PROGRAM RemovalProgram
VAR
END_VAR

// Written 25.8.2023 by Daniel Kelly

// The purpose of this POU is to automate the emptying of the system
//OpenValves will open both top and bottom valves
//RemovalMotorON will turn on the removal motor
//FM1_ON turns on the grey feeding motor M1
// The steps OFF1, OFF2 etc. turns of the removal motor and both top and bottom valves

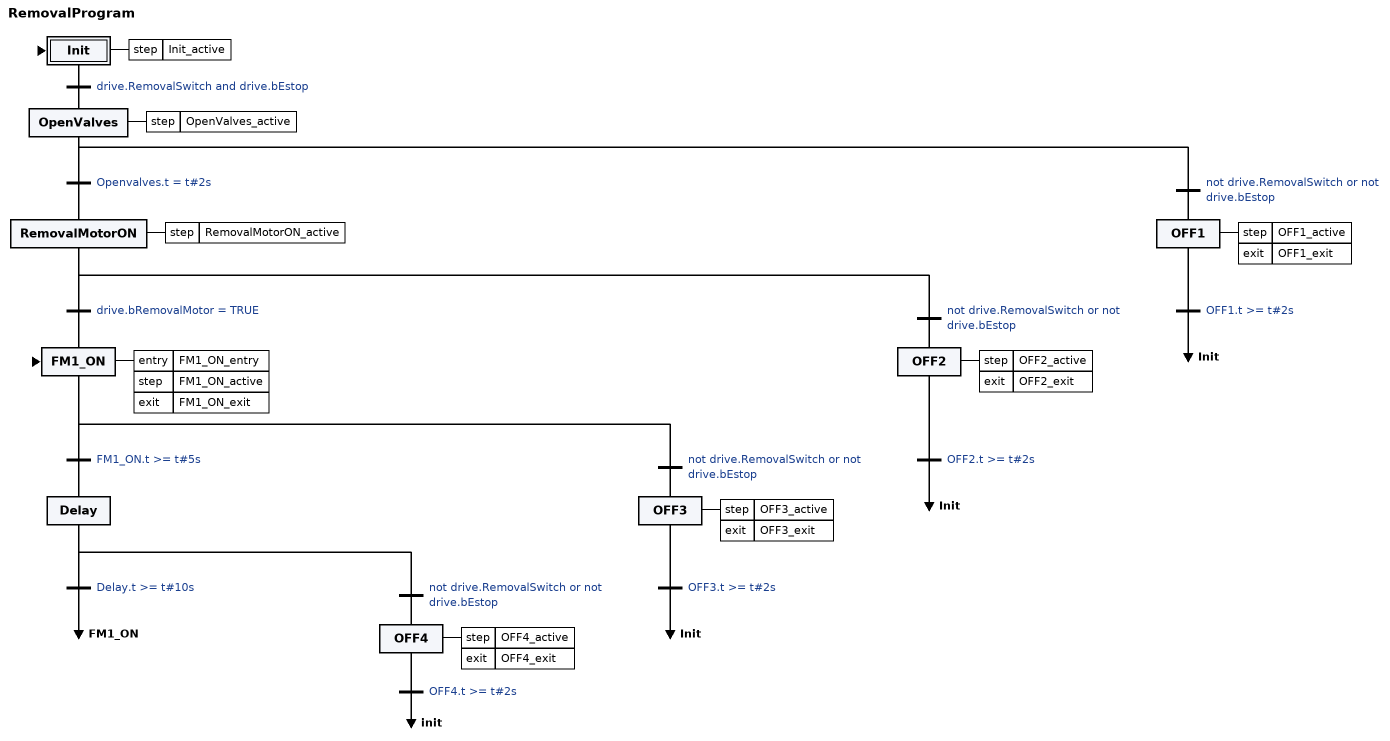
INITIAL_STEP Init:
    Init_active(N);  // step action
END_STEP
TRANSITION FROM Init TO OpenValves
    := drive.RemovalSwitch and drive.bEstop;
END_TRANSITION
STEP OpenValves:
    OpenValves_active(N);  // step action
END_STEP
TRANSITION FROM OpenValves TO RemovalMotorON
    := Openvalves.t = t#2s;
END_TRANSITION
TRANSITION FROM OpenValves TO OFF1
    := not drive.RemovalSwitch or not drive.bEstop;
END_TRANSITION
STEP OFF1:
    OFF1_active(N);  // step action
    OFF1_exit(P0);  // exit action
END_STEP
TRANSITION FROM OFF1 TO Init
    := OFF1.t >= t#2s;
END_TRANSITION
STEP RemovalMotorON:
    RemovalMotorON_active(N);  // step action
END_STEP
TRANSITION FROM RemovalMotorON TO FM1_ON
    := drive.bRemovalMotor = TRUE;
END_TRANSITION
TRANSITION FROM RemovalMotorON TO OFF2
    := not drive.RemovalSwitch or not drive.bEstop;
END_TRANSITION
STEP OFF2:
    OFF2_active(N);  // step action
    OFF2_exit(P0);  // exit action
END_STEP
TRANSITION FROM OFF2 TO Init
    := OFF2.t >= t#2s;
END_TRANSITION
STEP FM1_ON:
    FM1_ON_entry(P1);  // entry action
    FM1_ON_active(N);  // step action
    FM1_ON_exit(P0);  // exit action
END_STEP
TRANSITION FROM FM1_ON TO Delay
    := FM1_ON.t >= t#5s;
END_TRANSITION
TRANSITION FROM FM1_ON TO OFF3
    := not drive.RemovalSwitch or not drive.bEstop;
END_TRANSITION
STEP OFF3:
    OFF3_active(N);  // step action
    OFF3_exit(P0);  // exit action
END_STEP
TRANSITION FROM OFF3 TO Init
    := OFF3.t >= t#2s;
END_TRANSITION
STEP Delay:
END_STEP
TRANSITION FROM Delay TO FM1_ON
    := Delay.t >= t#10s;
END_TRANSITION
TRANSITION FROM Delay TO OFF4
    := not drive.RemovalSwitch or not drive.bEstop;
END_TRANSITION
STEP OFF4:
    OFF4_active(N);  // step action
    OFF4_exit(P0);  // exit action
END_STEP
TRANSITION FROM OFF4 TO init
    := OFF4.t >= t#2s;
END_TRANSITION

ACTION FM1_ON_active:
IF drive.ATV_TPDO_Input1_Status_Word = atv_status.rdy2SwitchON THEN 
	drive.ATV_RPDO_Output1_Control_Word := 7;
END_IF

IF drive.ATV_TPDO_Input1_Status_Word = atv_status.SwitchedON THEN 
	drive.ATV_RPDO_Output1_Control_Word := 15;
	
END_IF

drive.bM1active := TRUE;
END_ACTION

ACTION FM1_ON_entry:
drive.ATV_RPDO_Output2_Target_Velocity := 1000;
drive.ATV_RPDO_Output1_Control_Word := 6;
END_ACTION

ACTION FM1_ON_exit:
drive.ATV_RPDO_Output1_Control_Word := 7; 
drive.bM1active := FALSE;
END_ACTION

ACTION Init_active:

END_ACTION

ACTION OFF1_active:
drive.bRemovalMotor := FALSE;
drive.CloseTopValve := TRUE;
drive.CloseBottomValve := TRUE;

drive.OpenTopValve := FALSE;
drive.OpenBottomValve := FALSE;

drive.bValveLamp := FALSE;
END_ACTION

ACTION OFF1_exit:
drive.CloseBottomValve := FALSE;
drive.CloseTopValve := FALSE;
END_ACTION

ACTION OFF2_active:
drive.bRemovalMotor := FALSE;
drive.CloseTopValve := TRUE;
drive.CloseBottomValve := TRUE;

drive.OpenTopValve := FALSE;
drive.OpenBottomValve := FALSE;

drive.bValveLamp := FALSE;
END_ACTION

ACTION OFF2_exit:
drive.CloseBottomValve := FALSE;
drive.CloseTopValve := FALSE;
END_ACTION

ACTION OFF3_active:
drive.bRemovalMotor := FALSE;
drive.CloseTopValve := TRUE;
drive.CloseBottomValve := TRUE;

drive.OpenTopValve := FALSE;
drive.OpenBottomValve := FALSE;

drive.bValveLamp := FALSE;
drive.bM1active := FALSE;
END_ACTION

ACTION OFF3_exit:
drive.CloseBottomValve := FALSE;
drive.CloseTopValve := FALSE;
END_ACTION

ACTION OFF4_active:
drive.bRemovalMotor := FALSE;
drive.CloseTopValve := TRUE;
drive.CloseBottomValve := TRUE;

drive.OpenTopValve := FALSE;
drive.OpenBottomValve := FALSE;

drive.bValveLamp := false;
END_ACTION

ACTION OFF4_exit:
drive.CloseBottomValve := FALSE;
drive.CloseTopValve := FALSE;
END_ACTION

ACTION OpenValves_active:
drive.CloseTopValve := FALSE;
drive.CloseBottomValve := FALSE;


drive.OpenTopValve := TRUE;
drive.OpenBottomValve := TRUE;

drive.bValveLamp := TRUE;
END_ACTION

ACTION RemovalMotorON_active:
drive.bRemovalMotor := TRUE;
END_ACTION

ACTION TurnOFFValve_active:

END_ACTION

END_PROGRAM

(* stored: Version 1.1.0.1, ProductVersion 3.1.4024.12
   POU RemovalProgram: Id {ae0e60ad-094d-445a-b2f1-48070b107328}, SpecialFunc None
   Action FM1_ON_active: Id {aaa71c50-0c48-47dc-8cc2-1dd2bce4c1ca}
   Action FM1_ON_entry: Id {23893ef5-b789-4def-a398-69e638e5066d}
   Action FM1_ON_exit: Id {36a1cbb2-4829-49ae-b0e6-8da9386f9876}
   Action Init_active: Id {9db596b9-eaf7-4ad8-b8d4-8e77a339c298}
   Action OFF1_active: Id {1d1c81d8-26cf-4f71-97b7-38bb65c99d67}
   Action OFF1_exit: Id {30a16948-ebaa-42e4-87b9-5f785438d26e}
   Action OFF2_active: Id {c097a4f4-c8d1-4ac1-8241-0411b5728a52}
   Action OFF2_exit: Id {4b292cf5-f4fa-492c-aded-c886a2c35b93}
   Action OFF3_active: Id {fd07b831-02d0-4b03-b31e-cf7cd8d7568a}
   Action OFF3_exit: Id {585447f6-8641-455d-87c1-7ac825f06ba8}
   Action OFF4_active: Id {68de2a0f-46b8-40cf-ad33-d7c1f2f987d9}
   Action OFF4_exit: Id {4eda5a2c-f1c1-4ce5-a936-5b4096d1119d}
   Action OpenValves_active: Id {830ddc11-174b-45e2-bbd3-eef7d43ab51e}
   Action RemovalMotorON_active: Id {cf5af986-ee38-413d-9514-d19f4249a50f}
   Action TurnOFFValve_active: Id {81910142-97b4-413c-a669-087156d8e2ab} *)
